{attribute 'linkalways'}
{attribute 'no_explicit_call' := 'This FB is a CLASS and must be accessed using methods or properties'}
{attribute 'enable_dynamic_creation'}
FUNCTION_BLOCK Node_F_VN_InvertImageColorExp EXTENDS VisionNode
VAR
    ipSrcImage : _ITcVnImage;
    ipDestImage : _ITcVnImage;
    fMaxValue : _LREAL(-1);
    hrPrev : _HRESULT(S_OK);
    hresult : _HRESULT(S_OK);
END_VAR

METHOD PUBLIC Clone : I_Node
VAR
    pNode : POINTER TO Node_F_VN_InvertImageColorExp;
END_VAR
pNode := __NEW(Node_F_VN_InvertImageColorExp);
Clone := pNode^;
END_METHOD

METHOD FB_init : BOOL
VAR_INPUT
    bInitRetains : BOOL;
    bInCopyCode : BOOL;
END_VAR
AddInput('ipSrcImage', ipSrcImage);
AddOutput('ipDestImage', ipDestImage);
AddParameter('fMaxValue', fMaxValue);
AddInput('hrPrev', hrPrev);
AddOutput('hresult', hresult);
END_METHOD

METHOD PROTECTED OnExecute
hresult.Value := F_VN_InvertImageColorExp(
    ipSrcImage := ipSrcImage.Value,
    ipDestImage := ipDestImage.Value,
    fMaxValue := fMaxValue.Value,
    hrPrev := hrPrev.Value);
END_METHOD

METHOD PUBLIC PreExecutionCheck
VAR_INPUT
    Check : I_PreExecutionChecks;
END_VAR
Check.IsTrue(ipSrcImage.IsValid, 'ipSrcImage must contain an image');
END_METHOD

END_FUNCTION_BLOCK

(* stored: Version 1.1.0.1, ProductVersion 3.1.4026.25
   POU Node_F_VN_InvertImageColorExp: Id {edb4a322-5721-420f-b2e3-2a9d352f92e5}, SpecialFunc None
   Folder Constructor: Id {d52c45de-75d5-49d0-8dd2-b53786b31d4b}
   Method Clone: Id {746543c1-9c04-4c87-9ebb-928602aa8525}
   Method FB_init: Id {7cf6a78a-8621-4dcf-8e86-a19cb886c713}
   Method OnExecute: Id {1a51d332-cc4f-4ac0-93e0-023ddedefa80}
   Method PreExecutionCheck: Id {2b359882-7531-4dad-b91d-5ba5ebb45412} *)
